{attribute 'GeneratedUsingTerminal: EJ2521-0224-0016'}
{attribute addProperty BoxType "EJ2521-0224-0016"}
{attribute addProperty Id "StatusAT %I*Status_B83811715"}
{attribute addProperty CRC "3773501672"}
{attribute addProperty Size "5"}
TYPE PTO_Status_E0EB10E8 :
STRUCT
	{attribute addProperty Name "Status"}
	Status AT %I* : Status_B8381171;
END_STRUCT
END_TYPE

(* stored: Version 1.2.0.0, ProductVersion 3.1.4024.9
   DUT PTO_Status_E0EB10E8: Id {f146b3c6-8a79-41ed-b134-bd4c7fcb20a3} *)
